// TIA Portal V16 export
// export: Created 2022-02-04T14:40:23.4631666Z, ExportSetting WithDefaults, DisplayName Totally Integrated Automation Portal, DisplayVersion V16 Update 1, DisplayName TIA Portal Version Control Interface, DisplayVersion V16, DisplayName TIA Portal Openness, DisplayVersion V16, DisplayName SINAMICS Startdrive Advanced, DisplayVersion V16 Update 5, DisplayName SINAMICS Startdrive G130, G150, S120, S150, SINAMICS MV, S210, DisplayVersion V16 Update 5, DisplayName SINAMICS Startdrive G110M, G120, G120C, G120D, G120P, G115D, DisplayVersion V16 Update 5, DisplayName STEP 7 Professional, DisplayVersion V16, DisplayName STEP 7 Safety, DisplayVersion V16, DisplayName WinCC Advanced, DisplayVersion V16, DisplayName SIMATIC Visualization Architect, DisplayVersion V16
DATA_BLOCK "KeyFazer_Counter_DB"   // DB29
AUTHOR : Aspir
VERSION : 0.1
// stored: AutoNumber true, InstanceOfName KeyFazer_Counter, InstanceOfType FB
"KeyFazer_Counter"
   // VAR_INPUT
   //    NewWheel : Bool;
   //    RealChain : Bool;
   //    KeyFazerSignal : Bool;
   //    PlankSensor : Bool;
   //    AwaitedChain : Bool;
   //    Reset_count : Bool;
   //    Reset_alarms : Bool;
   //    PT : Int;
   // END_VAR
   // VAR_OUTPUT
   //    AlarmCount : Bool;
   //    Counted_one : Bool;
   // END_VAR
   // VAR_IN_OUT
   //    "Counter" : Int;
   // END_VAR
   // VAR RETAIN
   //    PlankCounted : Bool;
   //    PlankSensor_old : Bool;
   //    PlankSensor_filter : TON;
   // END_VAR
BEGIN
END_DATA_BLOCK
